(* IEC 61131-3 sources: Intern/plc_code, 3 files *)

(* ---- breaker.st ---- *)
PROGRAM ied_read
  VAR
    bus_voltage_0 AT %IW100 : INT;
    current_0 AT %IW101 : INT;
    line_cb_0 AT %QW100 : INT;
  END_VAR
  VAR
    test : BOOL := false;
    Tripvalue : INT := 1000;
  END_VAR

  IF bus_voltage_0 < 1000 THEN
    line_cb_0 := 1 - line_cb_0;
  END_IF;

END_PROGRAM

CONFIGURATION Config0
    RESOURCE Res0 ON PLC
        TASK Task0(INTERVAL := T#2000ms, PRIORITY := 0);
        PROGRAM Inst0 WITH Task0 : ied_read;
    END_RESOURCE
END_CONFIGURATION

(* ---- breaker_test.st ---- *)
PROGRAM ied_read
  VAR
    voltage AT %QW0 : INT;
    current AT %QW1 : INT;
    breaker AT %QW2 : INT;
  END_VAR
  VAR
    test : BOOL := false;
  END_VAR

  IF voltage > 100 THEN
    test := false;
  ELSE
    test := true;
  END_IF;

END_PROGRAM

CONFIGURATION Config0
    RESOURCE Res0 ON PLC
        TASK Task0(INTERVAL := T#10ms, PRIORITY := 1);
        PROGRAM Inst0 WITH Task0 : ied_read;
    END_RESOURCE
END_CONFIGURATION

(* ---- breaker_test_2.st ---- *)
PROGRAM read
  VAR
    a AT %MW0 : INT;
    b AT %MW1 : INT;
    c AT %MW2 : INT;
  END_VAR
  VAR
    test : BOOL := false;
    Tripvalue : INT := 1000;
  END_VAR

  c := 1;

END_PROGRAM

CONFIGURATION Config0
    RESOURCE Res0 ON PLC
        TASK Task0(INTERVAL := T#20ms, PRIORITY := 0);
        PROGRAM instance0 WITH task0 : read;
    END_RESOURCE
END_CONFIGURATION
